(* IEC 61131-3 sources: CodesysTest/export/Unused/FB_SimBasicBagDelivery.pou/BagSeparated.prop, 1 file *)

(* ---- Get.pm.st ---- *)
(*#-#-#-#-#-#-#-#-#-#---Declaration---#-#-#-#-#-#-#-#-#-#-#-#-#*)

VAR
END_VAR
(*#-#-#-#-#-#-#-#-#-#---Implementation---#-#-#-#-#-#-#-#-#-#-#-#-#*)

BagSeparated := reverseToSeparate.Q;
